PROGRAM POU
VAR
END_VAR

Conveyors.cfgP6005IntlksArry[0].Description := 'Panel E-Stop';
Conveyors.cfgP6005IntlksArry[0].DeviceLabel := 'PB1';
Conveyors.cfgP6005IntlksArry[0].OKState := TRUE;
Conveyors.cfgP6005IntlksArry[0].StopCode := E_StopCodes.SystemStop;




Conveyors.cfgP6005EvntsArry[0].Description := 'Panel E-Stop';
Conveyors.cfgP6005EvntsArry[0].DeviceLabel := 'PB1';
Conveyors.cfgP6005EvntsArry[0].OKState := TRUE;
Conveyors.cfgP6005EvntsArry[0].StopCode := E_StopCodes.SystemStop;

END_PROGRAM

(* stored: Version 1.1.0.1, ProductVersion 3.1.4024.4
   POU POU: Id {6cd5ee68-407e-4a34-8be8-ec30122f0457}, SpecialFunc None *)
